(* CODESYS project Functions.export

Project tree, tasks and I/O mapping:
  Functions/
    function F_TRMAddEventHandler [ST]
    function F_TRMReader [ST]
    function F_TRMSender [ST]
    function Real2Register [ST]
    function Register2Real [ST]
*)

// Functions/F_TRMAddEventHandler
FUNCTION F_TRMAddEventHandler : BOOL
VAR_INPUT
	refFIFO: POINTER TO FIFO.FIFO;
	Stage:	INT;
	refEvent: POINTER TO BOOL;
END_VAR
VAR_OUTPUT
	xError:		BOOL;
END_VAR
VAR
END_VAR

IF refFIFO^.isFull THEN
	xError:=TRUE;
	RETURN;
END_IF

refFIFO^.Push(Stage);
refEvent^:=FALSE;
xError:=FALSE;
RETURN;

END_FUNCTION

// Functions/F_TRMReader
FUNCTION F_TRMReader : BOOL
VAR_INPUT
	ptrStruct: 			POINTER TO BYTE; 	//Указатель на структуру для обхода
	uiStructureSize:	UINT;				//Размер структуры в байтах
	uiSize: 			UINT;				//Количество элементов в структуре.
	ptrReadInt:  			POINTER TO OwenNet.OWEN_GET_DINT;
	ptrReadFloat:			POINTER TO OwenNet.OWEN_GET_REAL;
	ptrReadOther:			POINTER TO owenNet.OWEN_UNI_IO;
END_VAR
VAR_OUTPUT
	xError: BOOL;
	Error:  WORD;
	Complete: BOOL;
END_VAR
VAR
	ptrUnit:	POINTER TO OwenValue;
	uiCount:	UINT;//Переменная счетчик для цикла
	iOperation:	INT;//Переменная для Switch case
	wError: WORD;
END_VAR

FOR uiCount:=0 TO uiSize-1 BY 1 DO
	ptrUnit:=ptrStruct+(SIZEOF(OwenValue)*uiCount);
	iOperation:=ptrUnit^.ValueType;
	CASE iOperation OF
		OWEN_TYPE.INTEGER:
			ptrReadInt^.Index:=ptrUnit^.ID;
			ptrReadInt^.IntType:=OwenNet.UINT_FRM;
			ptrReadInt^.Name:=ptrUnit^.ParameterName;
			ptrReadInt^.Value:=ptrUnit^.IntValue;
			ptrReadInt^(Enable:=TRUE);
			IF ptrReadInt^.Complete  OR ptrReadInt^.Error<>0 THEN
				
				IF ptrReadInt^.Error = 0 THEN
					ptrUnit^.IntValue:=ptrReadInt^.Value;
				END_IF
				ptrReadInt^(Enable:=FALSE);
				wError:=ptrReadInt^.Error;
			END_IF
		OWEN_TYPE.FLOAT:
			ptrReadFloat^.Index:=ptrUnit^.ID;
			ptrReadFloat^.RealType:=OwenNet.OW_FL32;
			ptrReadFloat^.Name:=ptrUnit^.ParameterName;
			ptrReadFloat^.Value:=ptrUnit^.FloatValue;
			ptrReadFloat^(Enable:=TRUE);
			IF ptrReadFloat^.Complete OR ptrReadFloat^.Error<>0 THEN
				IF ptrReadFloat^.Error = 0 THEN
					ptrUnit^.FloatValue:=ptrReadFloat^.Value;
				END_IF
				wError:=ptrReadFloat^.Error;
				ptrReadFloat^(Enable:=FALSE);
			END_IF	
	END_CASE
	IF wError<>0 THEN
		xError:=TRUE;
		Error:=wError;
		RETURN;
	END_IF
END_FOR
Complete:=TRUE;
return;

END_FUNCTION

// Functions/F_TRMSender
FUNCTION F_TRMSender : BOOL
VAR_INPUT
	ptrStruct: 			POINTER TO BYTE; 						//Указатель на структуру для обхода
	uiStructureSize:	UINT;									//Размер структуры в байтах
	uiSize: 			UINT;									//Количество элементов в структуре.
	ptrWriteInt:  			POINTER TO OwenNet.OWEN_SET_DINT; 	
	ptrWriteFloat:			POINTER TO OwenNet.OWEN_SET_REAL;		
	ptrWriteOther:			POINTER TO OwenNet.OWEN_UNI_IO;		
END_VAR
VAR_OUTPUT
	xError: BOOL;												//Error
	Error:  WORD;												//Error Status OwenNet
	Complete: BOOL;												//Process complete without error
END_VAR
VAR
	ptrUnit:	POINTER TO OwenValue;
	uiCount:	UINT;											//Переменная счетчик для цикла
	iOperation:	INT;											//Переменная для Switch case
	wError: WORD;
END_VAR

FOR uiCount:=0 TO uiSize-1 BY 1 DO
	ptrUnit:=ptrStruct+(SIZEOF(OwenValue)*uiCount);
	iOperation:=ptrUnit^.ValueType;
	CASE iOperation OF
		OWEN_TYPE.INTEGER:
			ptrWriteInt^.Index:=ptrUnit^.ID;
			ptrWriteInt^.IntType:=OwenNet.UINT_FRM;
			ptrWriteInt^.Name:=ptrUnit^.ParameterName;
			ptrWriteInt^.Value:=ptrUnit^.IntValue;
			ptrWriteInt^(Enable:=TRUE);
			IF ptrWriteInt^.Complete  OR ptrWriteInt^.Error<>0 THEN
				ptrWriteInt^(Enable:=FALSE);
				wError:=ptrWriteInt^.Error;
			END_IF
		
			
		OWEN_TYPE.FLOAT:
			ptrWriteFloat^.Index:=ptrUnit^.ID;
			ptrWriteFloat^.RealType:=OwenNet.OW_FL32;
			ptrWriteFloat^.Name:=ptrUnit^.ParameterName;
			ptrWriteFloat^.Value:=ptrUnit^.FloatValue;
			ptrWriteFloat^(Enable:=TRUE);
			IF ptrWriteFloat^.Complete OR ptrWriteFloat^.Error<>0 THEN
				ptrWriteFloat^(Enable:=FALSE);
				wError:=ptrWriteFloat^.Error;
			END_IF
			
		(*OWEN_TYPE.OTHER:
			WriteOther.Index:=ptrUnit^.ID;
			WriteOther.Name:=ptrUnit^.ParameterName;
			WriteOther.BufSize:=17;
			WriteOther.Buffer:=ptrUnit^.OtherValue;*)
	END_CASE
	IF wError<>0 THEN
		xError:=TRUE;
		Error:=wError;
		RETURN;
	END_IF
END_FOR
Complete:=TRUE;
RETURN;

END_FUNCTION

// Functions/Real2Register
FUNCTION Real2Register : UINT
VAR_INPUT
	rValue:				REAL;
	iPointPosition:		INT;
	
END_VAR
VAR
END_VAR

Real2Register:=REAL_TO_UINT(rValue*(EXPT(10,iPointPosition)));

END_FUNCTION

// Functions/Register2Real
FUNCTION Register2Real : REAL
VAR_INPUT
	uiRegister: UINT;
	iPointPosition: INT;
END_VAR
VAR
END_VAR

Register2Real:=((UINT_TO_REAL(uiRegister))/(EXPT(10.0,iPointPosition)));

END_FUNCTION
